// TIA Portal V19 export
TYPE "UDT_SIM_INT"
   STRUCT
      en : Bool;
      value : Int;
   END_STRUCT;
END_TYPE
